// TIA Portal project "FactoryIO_Template_S7-1200_V16_V16" (V16)
// Vorlageprojekt für das Buch mit Zielsystem S7-1200

(* hardware
DEVICE "S7-1200-Station_1"  S7-1200 Station
   slot 0: "Baugruppenträger_0"  Rack  V1.0
   slot 1: "PLC_1"  CPU 1211C DC/DC/DC  6ES7 211-1AE40-0XB0  V4.1
*)

// ===== PLC "PLC_1"  CPU 1211C DC/DC/DC =====

VAR_GLOBAL   // PLC tag table "Standard-Variablentabelle"
   "EMITTER" AT %A0.0 : Bool;
   "START" AT %E0.0 : Bool;
   "STOP" AT %E0.1 : Bool;
   "BELT 2M" AT %Q0.1 : Bool;
   "BELT 4M" AT %Q0.2 : Bool;
   "SENSOR 1" AT %I0.3 : Bool;
   "BELT 6M" AT %Q0.3 : Bool;
   "SENSOR 2" AT %I0.4 : Bool;
   "UP" AT %Q0.4 : Bool;
   "DOWN" AT %Q0.5 : Bool;
   "R LIMIT" AT %I0.2 : Bool;
   "L LIMIT" AT %I0.5 : Bool;
   "ELVATOR +" AT %Q0.6 : Bool;
   "MARKER 1" AT %M0.1 : Bool;
   "MARKER 2" AT %M0.2 : Bool;
   "MARKER 3" AT %M0.3 : Bool;
END_VAR

FUNCTION "MHJ-PLC-Lab-Function-S71200" : Void   // FC9000, SCL
{ S7_Optimized_Access := 'TRUE' }
VERSION : 0.1
   VAR_TEMP
      rdTimeReturn : Int;
      outputTime : DTL;
      SyncVal : Byte;
      forVal : Int;
      forVal_2 : Int;
      Value : Byte;
   END_VAR
   VAR CONSTANT
      CompVal : Byte := 16#34;
      Value_01 : Byte := 16#11;
      Value_01_DW : DWord := 16#A165_D992;
      Value_02_DW : DWord := 16#58BE_4401;
   END_VAR
BEGIN

   #Value:=PEEK(area := 16#82,
        dbNumber := 0,
        byteOffset := 511);
   #Value := #Value + 1;

   POKE(area := 16#82,
        dbNumber := 0,
        byteOffset := 511,
        value := #Value);

   POKE(area:=16#81,
        dbNumber:=0,
        byteOffset:=1016,
        value:=#Value_01_DW);
   POKE(area := 16#81,
        dbNumber := 0,
        byteOffset := 1020,
        value := #Value_02_DW);

   POKE(area := 16#81,
        dbNumber := 0,
        byteOffset := 511,
        value := B#16#00);

   FOR #forVal := 0 TO 120 DO
       FOR #forVal_2:=0 TO 10 DO
           #rdTimeReturn:=RD_SYS_T(#outputTime);
           #rdTimeReturn := WR_SYS_T(#outputTime);
           #rdTimeReturn := RD_SYS_T(#outputTime);
           #rdTimeReturn := WR_SYS_T(#outputTime);
       END_FOR;
       #SyncVal:= PEEK(area := 16#81,
                      dbNumber := 0,
                      byteOffset := 511);
       IF #SyncVal = #CompVal THEN
          GOTO M_1;
       END_IF;
   END_FOR;
   RETURN;

   M_1:
   POKE(area := 16#81,
        dbNumber := 0,
        byteOffset := 511,
        value := B#16#0);
END_FUNCTION

ORGANIZATION_BLOCK "Main"   // OB1, LAD, ProgramCycle
TITLE = "Main Program Sweep (Cycle)"
{ S7_Optimized_Access := 'TRUE' }
VERSION : 0.1
   VAR_INPUT
      Initial_Call : Bool;   // Initial call of this OB
      Remanence : Bool;   // =True, if remanent data are available
   END_VAR
   VAR_TEMP   // added for the SCL form of the ladder/FBD networks
      _w1 : Bool;
   END_VAR
BEGIN

REGION Network 1: Konnektierungsbaustein für PLC-Lab
   // Im Netzwerk 1 wird der Konnektierungsbaustein für PLC-Lab aufgerufen.
   // Dieser Aufruf darf nicht entfernt werden!
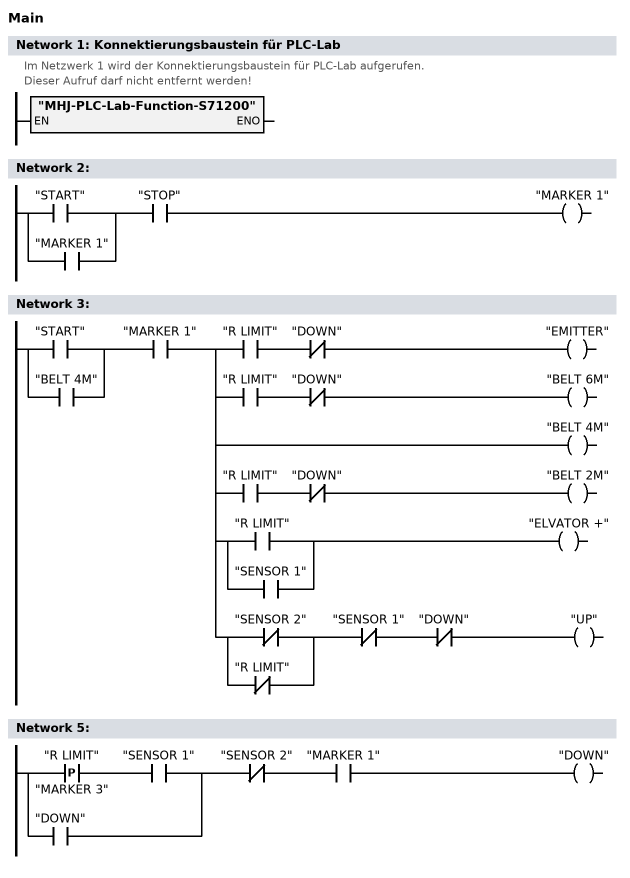
   RUNG wire#powerrail
      "MHJ-PLC-Lab-Function-S71200"()
   END_RUNG
   // the same network as SCL:
   "MHJ-PLC-Lab-Function-S71200"();
END_REGION

REGION Network 2
   RUNG wire#powerrail
      Contact( "START" )
      wire#w1
      Contact( "STOP" )
      Coil( "MARKER 1" )
   END_RUNG
   RUNG wire#powerrail
      Contact( "MARKER 1" )
   END_RUNG wire#w1
   // the same network as SCL:
   "MARKER 1" := ("START" OR "MARKER 1") AND "STOP";
END_REGION

REGION Network 3
   RUNG wire#powerrail
      Contact( "START" )
      wire#w1
      Contact( "MARKER 1" )
      wire#w2
      Contact( "R LIMIT" )
      I_Contact( "DOWN" )
      Coil( "EMITTER" )
   END_RUNG
   RUNG wire#powerrail
      Contact( "BELT 4M" )
   END_RUNG wire#w1
   RUNG wire#w2
      Contact( "R LIMIT" )
      I_Contact( "DOWN" )
      Coil( "BELT 6M" )
   END_RUNG
   RUNG wire#w2
      Coil( "BELT 4M" )
   END_RUNG
   RUNG wire#w2
      Contact( "R LIMIT" )
      I_Contact( "DOWN" )
      Coil( "BELT 2M" )
   END_RUNG
   RUNG wire#w2
      Contact( "R LIMIT" )
      wire#w3
      Coil( "ELVATOR +" )
   END_RUNG
   RUNG wire#w2
      Contact( "SENSOR 1" )
   END_RUNG wire#w3
   RUNG wire#w2
      I_Contact( "SENSOR 2" )
      wire#w4
      I_Contact( "SENSOR 1" )
      I_Contact( "DOWN" )
      Coil( "UP" )
   END_RUNG
   RUNG wire#w2
      I_Contact( "R LIMIT" )
   END_RUNG wire#w4
   // the same network as SCL:
   #_w1 := ("START" OR "BELT 4M") AND "MARKER 1";
   "EMITTER" := #_w1 AND "R LIMIT" AND NOT "DOWN";
   "BELT 6M" := #_w1 AND "R LIMIT" AND NOT "DOWN";
   "BELT 4M" := #_w1;
   "BELT 2M" := #_w1 AND "R LIMIT" AND NOT "DOWN";
   "ELVATOR +" := #_w1 AND ("R LIMIT" OR "SENSOR 1");
   "UP" := #_w1 AND (NOT "SENSOR 2" OR NOT "R LIMIT") AND NOT "SENSOR 1" AND NOT "DOWN";
END_REGION

REGION Network 5
   RUNG wire#powerrail
      P_Contact(operand := "R LIMIT", bit := "MARKER 3")
      Contact( "SENSOR 1" )
      wire#w1
      I_Contact( "SENSOR 2" )
      Contact( "MARKER 1" )
      Coil( "DOWN" )
   END_RUNG
   RUNG wire#powerrail
      Contact( "DOWN" )
   END_RUNG wire#w1
   // the same network as SCL:
   #_w1 := "R LIMIT" AND NOT "MARKER 3";   // rising edge of "R LIMIT"
   "MARKER 3" := "R LIMIT";
   "DOWN" := ((#_w1 AND "SENSOR 1") OR "DOWN") AND NOT "SENSOR 2" AND "MARKER 1";
END_REGION
END_ORGANIZATION_BLOCK